PROGRAM MAIN
VAR
	//Integrator
	ssMethodType : SINT := 1; 
	Timer : LREAL;
	
	//Pressure pA
	fbPressureGradient_pA : PressureGradient;
	PressurepA : LREAL;
	
	//Pressure pB
	fbPressureGradient_pB : PressureGradient;
	PressurepB : LREAL;
	
	//Pump
	fbPump : Pump;
	PumpTorque : LREAL;
	PumpFlowRate : LREAL;

	//OrificeEquation QA and QB
	fbOrificeEquationQA : OrificeEquation;
	fbOrificeEquationQB : OrificeEquation;	
	FlowQA : LREAL;
	FlowQB : LREAL;
	
	//HydraulicCylinder
	fbHydraulicCylinder : HydraulicCylinder;
	PressureBoreSide : LREAL;
	PressureRodSide : LREAL;
	AreaBoreSide : LREAL;
	AreaRodSide : LREAL;
	LoadForcePistonFL : LREAL;
	FrictionForce : LREAL;
	PistonMass : LREAL;
	
	pA : LREAL;
	pB : LREAL;
	qA : LREAL;
	qB : LREAL;
	ABore : LREAL;
	ARod : LREAL;
	xPos : LREAL;
	
END_VAR

//Timer
Timer := Timer + 0.01;

//Area Cylinder
ABore := EXPT(Param.DBore,2) * (Param.pi/4.0);
ARod := (EXPT(Param.DBore,2) - EXPT(Param.DRod,2)) * (Param.pi/4.0);

//Pump
fbPump(
	MotorSpeedRPM := 413.2,
	PumpDisplacement := 10.6E-6,
	DeltaMaxPressure := 250.0,
	PumpTorque => PumpTorque,
	PumpFlowRate => PumpFlowRate
	);
	
//Pressure Gradient pA and Pressure pA
fbPressureGradient_pA(
	TotalVolume := 2.9444E-04 + (fbHydraulicCylinder.PistonPosition * fbHydraulicCylinder.AreaBoreSide),
	BulkModulus := 10000.0,
	FlowrateIn := (FlowQA),
	FlowrateOut := (fbHydraulicCylinder.PistonVelocity * fbHydraulicCylinder.AreaBoreSide + 1),
	PressurePascal => PressurepA		//Pressure
	);
	
//Pressure Gradient pB and Pressure pB
fbPressureGradient_pB(
	TotalVolume := 2.9444E-04 + ((1.7 - fbHydraulicCylinder.PistonPosition) * fbHydraulicCylinder.AreaRodSide),
	BulkModulus := 10000.0,
	FlowrateIn := (fbHydraulicCylinder.PistonVelocity * fbHydraulicCylinder.AreaRodSide + 1),
	FlowrateOut := FlowQB,
	PressurePascal => PressurepB		//Pressure
	);


//OrificeEquationA (Q_A)
fbOrificeEquationQA(
	PressureOut := param.pT, 			//Found value from old simulink project, this one goes to the tank i guess
	PressureIn := PressurepA,		
	Kv := 0.5,
	ValveOpening := 1,	
	OrificeFlow => FlowQA
	);
	
//OrificeEquationB (Q_B)
fbOrificeEquationQB(
	PressureOut := param.pT, 			//Found value from old simulink project, this one goes to the tank i guess
	PressureIn := PressurepB,		
	Kv := 0.5,
	ValveOpening := 1,
	OrificeFlow => FlowQB
	);
	
//Hydraulic Cylinder 1
fbHydraulicCylinder(
	PistonMass := 5,
	LoadForcePistonFL := 1,
	FrictionForce := 1,
	AreaBoreSide := ABore,
	AreaRodSide := ARod,
	PressureBoreSide := PressurepA,
	PressureRodSide := PressurepB,
	PistonPosition => xPos
	);

END_PROGRAM

(* stored: Version 1.1.0.1, ProductVersion 3.1.4024.9
   POU MAIN: Id {d1c7ef4e-0337-49c7-9736-af80a39f1b25}, SpecialFunc None *)
